// TIA Portal V17 export
// export: Created 2025-01-08T13:55:35.2707621Z, ExportSetting WithDefaults, DisplayName Totally Integrated Automation Portal, DisplayVersion V17, DisplayName TIA Portal Openness, DisplayVersion V17, DisplayName TIA Portal Version Control Interface, DisplayVersion V17, DisplayName SINAMICS Startdrive Advanced, DisplayVersion V17 Update2, DisplayName SINAMICS Startdrive G130, G150, S120, S150, SINAMICS MV, S210, DisplayVersion V17 Update2, DisplayName SINAMICS Startdrive G110M, G120, G120C, G120D, G120P, G115D, DisplayVersion V17 Update2, DisplayName STEP 7 Professional, DisplayVersion V17, DisplayName STEP 7 Safety, DisplayVersion V17, DisplayName WinCC Advanced, DisplayVersion V17
DATA_BLOCK "DB - Motion_Settings"   // DB45
{ S7_Optimized_Access := 'FALSE' }
VERSION : 0.1
// stored: AutoNumber true, DBAccessibleFromOPCUA true, DBAccessibleFromWebserver true, IsOnlyStoredInLoadMemory false, IsWriteProtectedInAS false
   VAR RETAIN
      SideMotionSettings : Struct
         FeedLabelDistance : LReal := -700.0;
         FeedLabelVelocity : LReal := 2000.0;
         FeedLabelAcceleration : LReal := 30000.0;
         FeedLabelDeceleration : LReal := 30000.0;
         FeedLabelJerk : LReal := 1000000.0;
         DispenseLabelDistance : LReal := -675.0;
         DispenseLabelVelocity : LReal := 3000.0;
         DispenseLabelAcceleration : LReal := 500000.0;
         DispenseLabelDeceleration : LReal := 500000.0;
         DispenseLabelJerk : LReal := 5000000.0;
         DispenseLabelJerk_Stop : LReal := 5000000.0;
         DispenseLabelSensorCalibrationDistance : LReal := -84.0;
         RotateProductDistance : LReal := 900.0;
         RotateProductVelocity : LReal := -3000.0;
         RotateProductAcceleration : LReal := 50000.0;
         RotateProductDeceleration : LReal := 35000.0;
         RotateProductJerk : LReal := 2500000.0;
         IndexWheelDistance : LReal := -900.0;
         IndexWheelVelocity : LReal := 18000.0;
         IndexWheelAcceleration : LReal := 50000.0;
         IndexWheelDeceleration : LReal := 50000.0;
         IndexWheelJerk : LReal := 5000000.0;
         RewinderAcceleration : LReal := 20000.0;
         RewinderDeceleration : LReal := 30000.0;
         RewinderJerk : LReal := 2000000.0;
         RewinderPIDSetPoint : Real := 20.0;
         RewinderPIDGain : Real := 1.5;
         RewinderPIDIntegrationTime : Time := T#20s;
         RewinderPIDDeadZone : Real := 1.0;
         RewinderPIDOutputFactor : Real := 30.0;
      END_STRUCT;
      Zon1MotionSettings : Struct
         ConveyorVelocity : LReal := -1395.0;
         QueueVelocity : LReal := 140.0;
         SideHSMVelocity : LReal := 210.0;
         RotationRightRunningVelocity : LReal := 1500.0;
         RotationLeftRunningVelocity : LReal := -1500.0;
      END_STRUCT;
      Zon2MotionSettings : Struct
         ConveyorVelocity : LReal := -1395.0;
         QueueVelocity : LReal := -140.0;
         SideHSMVelocity : LReal := -210.0;
      END_STRUCT;
   END_VAR
BEGIN
END_DATA_BLOCK
